Fanuc TP program (LS listing): A_POS_CHANGE_BZG.LS

/PROG  A_POS_CHANGE_BZG
/ATTR
OWNER		= MNEDITOR;
COMMENT		= "";
PROG_SIZE	= 317;
CREATE		= DATE 25-11-18  TIME 20:32:44;
MODIFIED	= DATE 25-11-18  TIME 20:33:42;
FILE_NAME	= ;
VERSION		= 0;
LINE_COUNT	= 5;
MEMORY_SIZE	= 669;
PROTECT		= READ_WRITE;
TCD:  STACK_SIZE	= 0,
      TASK_PRIORITY	= 50,
      TIME_SLICE	= 0,
      BUSY_LAMP_OFF	= 0,
      ABORT_REQUEST	= 0,
      PAUSE_REQUEST	= 0;
DEFAULT_GROUP	= 1,*,*,*,*;
CONTROL_CODE	= 00000000 00000000;
/APPL
/APPL

AUTO_SINGULARITY_HEADER;
  ENABLE_SINGULARITY_AVOIDANCE   : TRUE;
  CYCLE_REFERENCE = 0, 0, 0, 0, 0, 0, 0, 0, 0, 0, 0, 0;
  CYCLE_TARGET =   0.00 ;
/MN
   1:  UFRAME_NUM=0 ;
   2:  UTOOL_NUM=1 ;
   3:   ;
   4:  PR[67,3:View pos offset]=PR[67,3:View pos offset]-40    ;
   5:   ;
/POS
/END
